// TIA Portal V17 export
// export: Created 2025-08-05T09:36:02.136916Z, ExportSetting WithDefaults, DisplayName Totally Integrated Automation Portal, DisplayVersion V17, DisplayName TIA Portal Openness, DisplayVersion V17, DisplayName TIA Portal Version Control Interface, DisplayVersion V17, DisplayName SINAMICS Startdrive Advanced, DisplayVersion V17, DisplayName SINAMICS Startdrive G130, G150, S120, S150, SINAMICS MV, S210, DisplayVersion V17, DisplayName SINAMICS Startdrive G110M, G120, G120C, G120D, G120P, G115D, DisplayVersion V17, DisplayName STEP 7 Professional, DisplayVersion V17, DisplayName STEP 7 Safety, DisplayVersion V17, DisplayName WinCC Advanced, DisplayVersion V17
TYPE "LaserComm_DDO"
// stored: IsFailsafeCompliant false
   STRUCT
      Valid : Bool;   // Data Loaded from Laser Comm and is Valid
      Min : Real;   // Minimum Point Value from LDD Measurement
      Max : Real;   // Maximum Point Value from LDD Measurement
      Mean : Real;   // Average Point Value from LDD Measurement
      Dev : Real;   // Standard Deviation of LDD Measurement
   END_STRUCT;
END_TYPE
